SUBAPPLICATION Uebung_010f3 (* SoftKey_F1 ODER AuxFunction2_X1 auf DigitalOutput_Q1 mit GreenWhiteBackground (SoftKey UND Aux) *)
  (* Standard: 61499-2; Description: Copyright (c) 2026 Meisterschulen am Ostbahnhof This program and the accompanying materials are made available under the terms of the Eclipse Public License 2.0 which is available at https://www.eclipse.org/legal/epl-2.0/ SPDX-License-Identifier: EPL-2.0 *)
  (* Version 1.0, 2026-09-06, Franz Höpfinger, Meisterschulen am Ostbahnhof, initial API and implementation and/or initial documentation *)
  PACKAGE Uebungen;
  IMPORT Uebungen::const::UT::DefaultPool::SoftKey_F1;
  IMPORT Uebungen::const::UT::DefaultPool::AuxFunction2_X1;
  IMPORT logiBUS::io::DQ::logiBUS_DO::Output_Q1;
  (* Documentation:
  SoftKey_F1 ODER AuxFunction2_X1 auf DigitalOutput_Q1 mit GreenWhiteBackground
   Kombiniert Uebung_010c (SoftKey mit Background) und Uebung_010f (Aux mit Background) auf einen gemeinsamen Ausgang: dieselbe Funktion ist sowohl über den VT-SoftKey als auch über den physischen Aux-Taster/Joystick bedienbar.
   Funktionsbeschreibung
    - SoftKey_F1 und AuxFunction2_X1 liefern je ein boolesches Signal, OR_2 verknüpft beide per ODER zu einem gemeinsamen Signal für DigitalOutput_Q1.
   - GreenWhiteBackground3 statt zwei einzelner GreenWhiteBackground1/GreenWhiteBackground2: dieser Baustein nimmt genau einen normalen VT-Objekt-Parameter (u16ObjId = SoftKey) UND einen Aux-Objekt-Parameter (u16ObjIdA = Aux) entgegen und setzt beide Hintergründe aus einem einzigen DI1-Eingang.
    Arbeitsauftrag
   Testen Sie: SoftKey_F1 drücken → Q1 EIN, beide Hintergründe (SoftKey und Aux) werden grün. Aux-Taster drücken → dasselbe. Werden beide gleichzeitig gehalten, bleibt Q1 EIN, bis beide losgelassen sind - Q1 schaltet erst AUS, wenn sowohl SoftKey_F1 als auch AuxFunction2_X1 wieder FALSE sind (reine ODER-Verknüpfung, kein Latch).
  *)
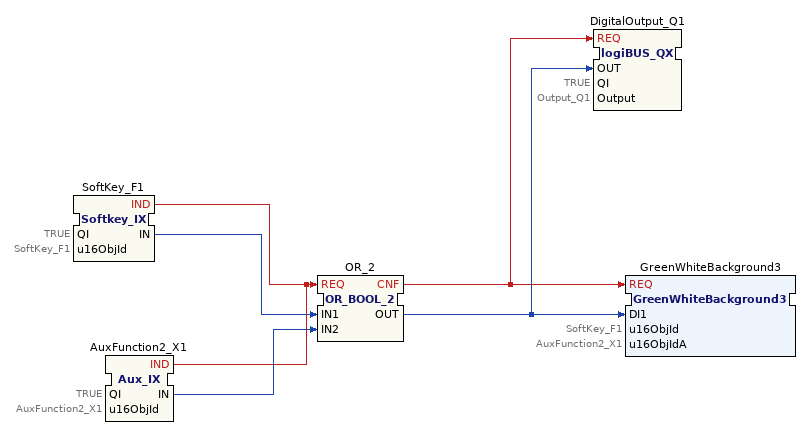
  (* SoftKey_F1 (VT) und AuxFunction2_X1 (Joystick) steuern denselben Q1 - ODER-verknuepft ueber OR_2. GreenWhiteBackground3 (nicht 1/2 einzeln!) bedient beide Hintergruende aus einem Baustein: u16ObjId=SoftKey (VT) und u16ObjIdA=Aux (VT+Aux-Handle). *)
  FBS
    DigitalOutput_Q1 : logiBUS::io::DQ::logiBUS_QX(QI := TRUE, Output := Output_Q1);
    SoftKey_F1 : isobus::UT::io::Softkey::Softkey_IX(QI := TRUE, u16ObjId := SoftKey_F1);
    AuxFunction2_X1 : isobus::UT::io::Auxiliary::IN::Aux_IX(QI := TRUE, u16ObjId := AuxFunction2_X1);
    OR_2 : iec61131::booleanOperators::OR_BOOL_2;
  END_FBS
  SUBAPPS
    GreenWhiteBackground3 : MyLib::sys::GreenWhiteBackground3(u16ObjId := SoftKey_F1, u16ObjIdA := AuxFunction2_X1);
  END_SUBAPPS
  EVENT_CONNECTIONS
    SoftKey_F1.IND TO OR_2.REQ;
    AuxFunction2_X1.IND TO OR_2.REQ;
    OR_2.CNF TO DigitalOutput_Q1.REQ;
    OR_2.CNF TO GreenWhiteBackground3.REQ;
  END_CONNECTIONS
  DATA_CONNECTIONS
    SoftKey_F1.IN TO OR_2.IN1;
    AuxFunction2_X1.IN TO OR_2.IN2;
    OR_2.OUT TO DigitalOutput_Q1.OUT;
    OR_2.OUT TO GreenWhiteBackground3.DI1;
  END_CONNECTIONS
END_SUBAPPLICATION
